(* PLC project Unnamed, Unknown Unnamed 1 *)
(* stored: creationDateTime 2026-08-07T23:20:52, modificationDateTime 2026-08-07T23:20:52 *)

PROGRAM main
  VAR_INPUT
    IceRequest : BOOL;
    MixType1 : BOOL;
    MixType2 : BOOL;
    MixType3 : BOOL;
    Liqueur1 : BOOL;
    Liqueur2 : BOOL;
    WaterRequest : BOOL;
  END_VAR
  VAR_OUTPUT
    DispenseIce : BOOL;
    DispenseMix1 : BOOL;
    DispenseMix2 : BOOL;
    DispenseMix3 : BOOL;
    DispenseLiqueur1 : BOOL;
    DispenseLiqueur2 : BOOL;
    DispenseWater : BOOL;
    CocktailReady : BOOL;
  END_VAR

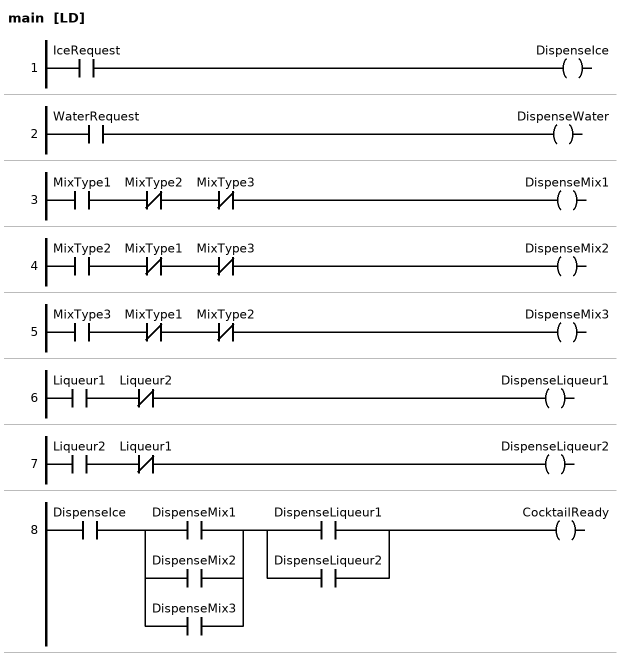
(* LD diagram, written out as Structured Text *)
DispenseIce := IceRequest;
DispenseWater := WaterRequest;
DispenseMix1 := MixType1 AND NOT MixType2 AND NOT MixType3;
DispenseMix2 := MixType2 AND NOT MixType1 AND NOT MixType3;
DispenseMix3 := MixType3 AND NOT MixType1 AND NOT MixType2;
DispenseLiqueur1 := Liqueur1 AND NOT Liqueur2;
DispenseLiqueur2 := Liqueur2 AND NOT Liqueur1;
CocktailReady := DispenseIce AND (DispenseMix1 OR DispenseMix2 OR DispenseMix3) AND (DispenseLiqueur1 OR DispenseLiqueur2);
END_PROGRAM

CONFIGURATION Config0
  RESOURCE Res0 ON PLC
    TASK task0(INTERVAL := T#20ms, PRIORITY := 1);
    PROGRAM instance0 WITH task0 : main;
  END_RESOURCE
END_CONFIGURATION
